DATA_BLOCK "DB_executeQuery"
{ S7_Optimized_Access := 'TRUE' }
VERSION : 0.1
NON_RETAIN
"FB_ExecuteQuery"

BEGIN

END_DATA_BLOCK

